Fanuc KAREL source: INIT_QUEUE.kl

PROGRAM T
%NOLOCKGROUP
VAR
 v0 : QUEUE_TYPE
BEGIN
 INIT_QUEUE(v0)
END T
